{attribute 'qualified_only'}
{attribute 'strict'}
TYPE E_DoorPos :
(
	UP,
	DOWN,
	UNDEFINED
);
END_TYPE

(* stored: Version 1.1.0.1, ProductVersion 3.1.4024.9
   DUT E_DoorPos: Id {b69eac6c-aa4a-47b8-aa7d-61ea297d94a5} *)
